// TIA Portal V20 export
FUNCTION_BLOCK "FB_AutoReset"   // FB21, LAD
// stored: Access Published, MemoryReserve 100, Namespace Global, SetENOAutomatically false
   VAR_INPUT
      AckIN : Bool;
   END_VAR
   VAR_OUTPUT
      Ack : Bool;
   END_VAR
   VAR
      MemoryBit : Array[1..2] of Bool;
      "Timer" { S7_SetPoint := 'True'} : TOF_TIME;
   END_VAR
   VAR_TEMP   // added for the SCL form of the ladder/FBD networks
      _w1 : Bool;
      _w2 : Bool;
   END_VAR
BEGIN

REGION Network 1
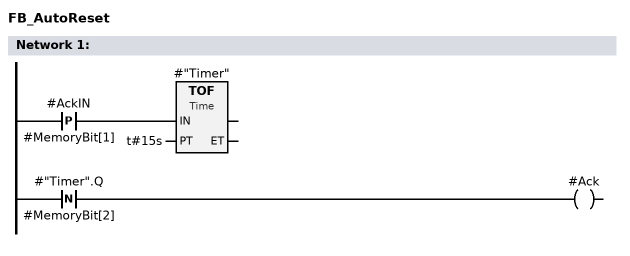
   RUNG wire#powerrail
      P_Contact(operand := #AckIN, bit := #MemoryBit[1])
      { S7_Templates := "time_type := Time" } #"Timer".TOF(pt := t#15s, et =>)
   END_RUNG
   RUNG wire#powerrail
      N_Contact(operand := #"Timer".Q, bit := #MemoryBit[2])
      Coil( #Ack )
   END_RUNG
   // the same network as SCL:
   #_w1 := #AckIN AND NOT #MemoryBit[1];   // rising edge of #AckIN
   #MemoryBit[1] := #AckIN;
   #"Timer"(IN := #_w1, PT := t#15s);   // TOF
   #_w2 := NOT #"Timer".Q AND #MemoryBit[2];   // falling edge of #"Timer".Q
   #MemoryBit[2] := #"Timer".Q;
   #Ack := #_w2;
END_REGION
END_FUNCTION_BLOCK
